(* IEC 61131-3 sources: matiec/benchmarks, 5 files *)

(* ---- b1_esd.st ---- *)
(* B1: Emergency Shutdown Interlock
 * Constructs: AND, OR, NOT, IF/ELSIF/ELSE, SR, TON, BOOL assignment
 * Scenario: Three trip sensors trigger an SR-latched alarm with TON delay.
 *           Manual acknowledge resets the latch.
 *)

PROGRAM esd_interlock
  VAR
    (* Inputs *)
    pressure_high  : BOOL;
    temp_high      : BOOL;
    flow_low       : BOOL;
    manual_reset   : BOOL;

    (* Internal *)
    any_trip       : BOOL;
    alarm_latch    : SR;
    alarm_delay    : TON;
    alarm_active   : BOOL;
    latched        : BOOL;

    (* Outputs *)
    shutdown_cmd   : BOOL;
    alarm_out      : BOOL;
  END_VAR

  (* Combine trip conditions: any single trip is enough *)
  any_trip := pressure_high OR temp_high OR flow_low;

  (* SR latch: Set on trip, Reset on manual acknowledge *)
  alarm_latch(S1 := any_trip, R := manual_reset);
  latched := alarm_latch.Q1;

  (* Delay alarm output by 3 seconds to filter transients *)
  alarm_delay(IN := latched, PT := T#3s);

  (* Output logic *)
  IF latched AND alarm_delay.Q THEN
    (* Confirmed alarm: shutdown and alarm *)
    shutdown_cmd := TRUE;
    alarm_out := TRUE;
  ELSIF latched AND NOT alarm_delay.Q THEN
    (* Alarm pending confirmation *)
    shutdown_cmd := FALSE;
    alarm_out := FALSE;
  ELSE
    (* No alarm *)
    shutdown_cmd := FALSE;
    alarm_out := FALSE;
  END_IF;

END_PROGRAM

CONFIGURATION esd_config
  RESOURCE esd_resource ON PLC
    TASK esd_task(INTERVAL := T#10ms, PRIORITY := 0);
    PROGRAM esd_inst WITH esd_task : esd_interlock;
  END_RESOURCE
END_CONFIGURATION

(* ---- b2_bms.st ---- *)
(* B2: Burner Management Purge Sequence
 * Constructs: R_TRIG, F_TRIG, TON (x2), INT state machine, nested ELSIF,
 *             INT comparison (=, <>), BOOL assignment
 * Scenario: 5-stage burner: idle(0)->purge(1)->ignite(2)->run(3)->lockout(4)
 *)

PROGRAM bms_purge
  VAR
    (* Inputs *)
    start_cmd      : BOOL;
    flame_sensor   : BOOL;
    purge_ok       : BOOL;

    (* State *)
    stage          : INT := 0;

    (* Edge detection *)
    start_edge     : R_TRIG;
    flame_lost     : F_TRIG;

    (* Timers *)
    purge_timer    : TON;
    ignition_timer : TON;

    (* Outputs *)
    fan_on         : BOOL;
    fuel_valve     : BOOL;
    igniter_on     : BOOL;
    alarm_lockout  : BOOL;
  END_VAR

  (* Detect start command rising edge *)
  start_edge(CLK := start_cmd);

  (* Detect flame loss falling edge *)
  flame_lost(CLK := flame_sensor);

  (* Purge timer: 30s air purge before ignition *)
  purge_timer(IN := (stage = 1), PT := T#30s);

  (* Ignition timer: 5s window to establish flame *)
  ignition_timer(IN := (stage = 2), PT := T#5s);

  (* State machine *)
  IF stage = 0 THEN
    (* IDLE *)
    fan_on := FALSE;
    fuel_valve := FALSE;
    igniter_on := FALSE;
    alarm_lockout := FALSE;
    IF start_edge.Q THEN
      stage := 1;
    END_IF;

  ELSIF stage = 1 THEN
    (* PURGE: fan on, wait 30s *)
    fan_on := TRUE;
    fuel_valve := FALSE;
    igniter_on := FALSE;
    IF purge_timer.Q AND purge_ok THEN
      stage := 2;
    END_IF;

  ELSIF stage = 2 THEN
    (* IGNITE: fan + fuel + igniter, 5s window *)
    fan_on := TRUE;
    fuel_valve := TRUE;
    igniter_on := TRUE;
    IF flame_sensor THEN
      stage := 3;
    ELSIF ignition_timer.Q AND NOT flame_sensor THEN
      stage := 4;
    END_IF;

  ELSIF stage = 3 THEN
    (* RUN: fan + fuel, monitor flame *)
    fan_on := TRUE;
    fuel_valve := TRUE;
    igniter_on := FALSE;
    IF flame_lost.Q THEN
      stage := 4;
    END_IF;

  ELSIF stage = 4 THEN
    (* LOCKOUT: everything off, alarm *)
    fan_on := FALSE;
    fuel_valve := FALSE;
    igniter_on := FALSE;
    alarm_lockout := TRUE;
    (* Require operator reset - not modeled here *)

  END_IF;

END_PROGRAM

CONFIGURATION bms_config
  RESOURCE bms_resource ON PLC
    TASK bms_task(INTERVAL := T#20ms, PRIORITY := 0);
    PROGRAM bms_inst WITH bms_task : bms_purge;
  END_RESOURCE
END_CONFIGURATION

(* ---- b3_conveyor.st ---- *)
(* B3: Conveyor with Part Counter
 * Constructs: CTU, R_TRIG, FOR loop (bounded), +, >, >=,
 *             boolean latch, INT arithmetic, BOOL assignment
 * Scenario: Conveyor counts parts via CTU. FOR loop computes batch totals.
 *)

PROGRAM conveyor_count
  VAR
    (* Inputs *)
    part_detect    : BOOL;
    batch_reset    : BOOL;
    run_cmd        : BOOL;
    batch_size     : INT := 10;

    (* Internal *)
    part_edge      : R_TRIG;
    part_counter   : CTU;
    motor_latch    : BOOL;
    batch_total    : INT := 0;
    idx            : INT;

    (* Outputs *)
    motor_on       : BOOL;
    batch_complete : BOOL;
    total_count    : INT;
  END_VAR

  (* Detect rising edge of part sensor *)
  part_edge(CLK := part_detect);

  (* Count parts: reset on batch_reset, target = batch_size *)
  part_counter(CU := part_edge.Q, R := batch_reset, PV := batch_size);

  (* Motor latch: start on run_cmd, stop on batch complete *)
  IF run_cmd THEN
    motor_latch := TRUE;
  END_IF;
  IF part_counter.Q THEN
    motor_latch := FALSE;
  END_IF;
  motor_on := motor_latch;

  (* Batch complete when counter reaches target *)
  batch_complete := part_counter.Q;
  total_count := part_counter.CV;

  (* Accumulate batch totals using FOR loop (5 batches) *)
  IF batch_complete THEN
    batch_total := 0;
    FOR idx := 1 TO 5 DO
      batch_total := batch_total + batch_size;
    END_FOR;
  END_IF;

END_PROGRAM

CONFIGURATION conveyor_config
  RESOURCE conveyor_resource ON PLC
    TASK conveyor_task(INTERVAL := T#10ms, PRIORITY := 0);
    PROGRAM conveyor_inst WITH conveyor_task : conveyor_count;
  END_RESOURCE
END_CONFIGURATION

(* ---- b4_shutdown.st ---- *)
(* B4: Multi-Stage Shutdown Sequence
 * Constructs: TON (x3), INT state machine, subtraction, < comparison,
 *             arithmetic (valve_pos - 10), IF/ELSIF chain
 * Scenario: 4-stage shutdown: running(0)->cooldown(1)->depressure(2)->safe(3)
 *           Each stage has a timer; valve position decrements per stage.
 *)

PROGRAM shutdown_seq
  VAR
    (* Inputs *)
    shutdown_req   : BOOL;

    (* State *)
    stage          : INT := 0;
    valve_pos      : INT := 100;

    (* Timers - one per stage *)
    cooldown_tmr   : TON;
    depress_tmr    : TON;
    safe_tmr       : TON;

    (* Outputs *)
    heater_on      : BOOL;
    pump_on        : BOOL;
    vent_open      : BOOL;
    safe_state     : BOOL;
  END_VAR

  (* Timer activations tied to current stage *)
  cooldown_tmr(IN := (stage = 1), PT := T#10s);
  depress_tmr(IN := (stage = 2), PT := T#15s);
  safe_tmr(IN := (stage = 3), PT := T#5s);

  IF stage = 0 THEN
    (* RUNNING: normal operation *)
    heater_on := TRUE;
    pump_on := TRUE;
    vent_open := FALSE;
    safe_state := FALSE;
    IF shutdown_req THEN
      stage := 1;
      valve_pos := 100;
    END_IF;

  ELSIF stage = 1 THEN
    (* COOLDOWN: heater off, pump still on *)
    heater_on := FALSE;
    pump_on := TRUE;
    vent_open := FALSE;
    valve_pos := valve_pos - 10;
    IF valve_pos < 0 THEN
      valve_pos := 0;
    END_IF;
    IF cooldown_tmr.Q THEN
      stage := 2;
    END_IF;

  ELSIF stage = 2 THEN
    (* DEPRESSURIZE: pump off, vent open *)
    heater_on := FALSE;
    pump_on := FALSE;
    vent_open := TRUE;
    valve_pos := valve_pos - 10;
    IF valve_pos < 0 THEN
      valve_pos := 0;
    END_IF;
    IF depress_tmr.Q THEN
      stage := 3;
    END_IF;

  ELSIF stage = 3 THEN
    (* SAFE: everything off *)
    heater_on := FALSE;
    pump_on := FALSE;
    vent_open := FALSE;
    safe_state := TRUE;
    IF safe_tmr.Q THEN
      (* Remain in safe state *)
      stage := 3;
    END_IF;

  END_IF;

END_PROGRAM

CONFIGURATION shutdown_config
  RESOURCE shutdown_resource ON PLC
    TASK shutdown_task(INTERVAL := T#50ms, PRIORITY := 0);
    PROGRAM shutdown_inst WITH shutdown_task : shutdown_seq;
  END_RESOURCE
END_CONFIGURATION

(* ---- b5_stress.st ---- *)
(* B5: WCET Stress - Synthetic Benchmark
   Exercises ALL LowPLC constructs: SR, RS, CTU, CTD, CTUD,
   TON, TOF, R_TRIG, F_TRIG, FOR loop, nested IF/ELSIF/ELSE,
   all comparison ops: EQ, NE, LT, GT, LE, GE,
   all arithmetic ops: ADD, SUB, MUL,
   all boolean ops: AND, OR, NOT, XOR.
   Uses inp_ prefix to avoid IN keyword collision. *)

PROGRAM stress_test
  VAR
    (* Inputs — use inp_ prefix since IN is a keyword *)
    inp_a          : BOOL;
    inp_b          : BOOL;
    inp_c          : BOOL;
    inp_d          : BOOL;
    inp_e          : INT := 0;
    inp_f          : INT := 50;
    inp_g          : INT := 100;
    inp_h          : TIME := T#2s;

    (* FB instances — all 9 standard FB types *)
    fb_sr          : SR;
    fb_rs          : RS;
    fb_ctu         : CTU;
    fb_ctd         : CTD;
    fb_ctud        : CTUD;
    fb_ton         : TON;
    fb_tof         : TOF;
    fb_rtrig       : R_TRIG;
    fb_ftrig       : F_TRIG;

    (* Working variables *)
    bool_res       : BOOL;
    int_res        : INT := 0;
    sum_acc        : INT := 0;
    idx            : INT;
    cmp_eq         : BOOL;
    cmp_ne         : BOOL;
    cmp_lt         : BOOL;
    cmp_gt         : BOOL;
    cmp_le         : BOOL;
    cmp_ge         : BOOL;

    (* Outputs *)
    out_alarm      : BOOL;
    out_count      : INT;
    out_timer_q    : BOOL;
    out_result     : INT;
  END_VAR

  (* --- Edge detectors --- *)
  fb_rtrig(CLK := inp_a);
  fb_ftrig(CLK := inp_b);

  (* --- Bistable latches --- *)
  fb_sr(S1 := fb_rtrig.Q, R := inp_c);
  fb_rs(S := inp_a, R1 := inp_d);

  (* --- Counters --- *)
  fb_ctu(CU := fb_rtrig.Q, R := inp_c, PV := inp_f);
  fb_ctd(CD := fb_ftrig.Q, LD := inp_d, PV := inp_g);
  fb_ctud(CU := inp_a, CD := inp_b, R := inp_c, LD := inp_d, PV := inp_f);

  (* --- Timers --- *)
  fb_ton(IN := fb_sr.Q1, PT := inp_h);
  fb_tof(IN := fb_rs.Q1, PT := T#1s);

  (* --- All comparison operators --- *)
  cmp_eq := (inp_e = inp_f);
  cmp_ne := (inp_e <> inp_f);
  cmp_lt := (inp_e < inp_f);
  cmp_gt := (inp_e > inp_f);
  cmp_le := (inp_e <= inp_f);
  cmp_ge := (inp_e >= inp_f);

  (* --- All boolean operators --- *)
  bool_res := (inp_a AND inp_b) OR (NOT inp_c) XOR inp_d;

  (* --- Arithmetic operators --- *)
  int_res := (inp_e + inp_f) - inp_g;
  int_res := int_res * 2;

  (* --- FOR loop with accumulator --- *)
  sum_acc := 0;
  FOR idx := 0 TO 9 DO
    sum_acc := sum_acc + idx;
  END_FOR;

  (* --- Nested IF/ELSIF/ELSE --- *)
  IF fb_ton.Q AND cmp_gt THEN
    out_alarm := TRUE;
    out_result := sum_acc + int_res;
  ELSIF fb_ctu.Q OR cmp_eq THEN
    out_alarm := FALSE;
    out_result := fb_ctu.CV + fb_ctd.CV;
  ELSIF cmp_le AND NOT cmp_ne THEN
    out_alarm := bool_res;
    out_result := fb_ctud.CV;
  ELSE
    out_alarm := FALSE;
    out_result := 0;
  END_IF;

  out_count := fb_ctu.CV;
  out_timer_q := fb_ton.Q;

END_PROGRAM

CONFIGURATION stress_config
  RESOURCE stress_resource ON PLC
    TASK stress_task(INTERVAL := T#10ms, PRIORITY := 0);
    PROGRAM stress_inst WITH stress_task : stress_test;
  END_RESOURCE
END_CONFIGURATION
